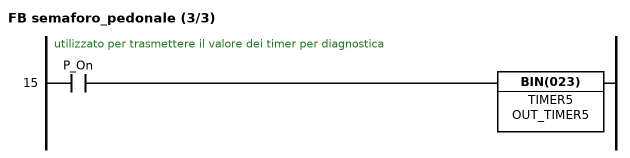
; [picture p24: FB semaforo_pedonale, rungs 15-15]
; rung 15: utilizzato per trasmettere il valore dei timer per diagnostica
LD P_On
BIN(023) TIMER5 OUT_TIMER5

## Function block stella_triangolo_MAT
VAR_INPUT
  start : BOOL;
  STOP : BOOL;
  ausiliario_K1 : BOOL;
  ausiliario_K2 : BOOL;
  ausiliario_K3 : BOOL;
  termica : BOOL;
  emergenza : BOOL;
END_VAR
VAR_OUTPUT
  linea : BOOL;
  stella : BOOL;
  triangolo : BOOL;
  lamp_blu : BOOL;
  lamp_verde1 : BOOL;
  lamp_verde2 : BOOL;
  lamp_gialla : BOOL;
  OUT_TIMER2 : WORD;
  OUT_TIMER1 : WORD;
END_VAR
VAR
  TIME : TIMER;
  err : BOOL;
END_VAR

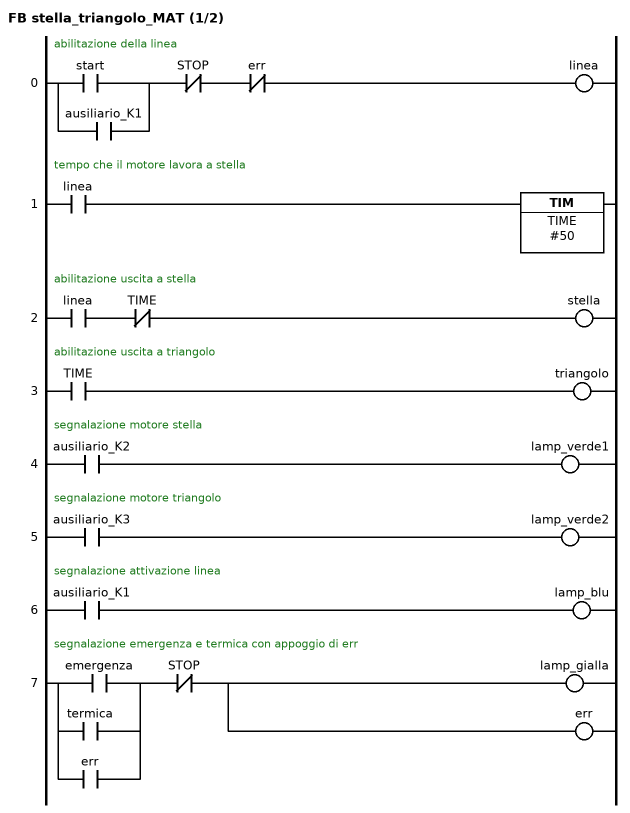
; rung 0: abilitazione della linea
LD start
OR ausiliario_K1
ANDNOT STOP
ANDNOT err
OUT linea
; rung 1: tempo che il motore lavora a stella
LD linea
TIM TIME #50
; rung 2: abilitazione uscita a stella
LD linea
ANDNOT TIME
OUT stella
; rung 3: abilitazione uscita a triangolo
LD TIME
OUT triangolo
; rung 4: segnalazione motore stella
LD ausiliario_K2
OUT lamp_verde1
; rung 5: segnalazione motore triangolo
LD ausiliario_K3
OUT lamp_verde2
; rung 6: segnalazione attivazione linea
LD ausiliario_K1
OUT lamp_blu
; rung 7: segnalazione emergenza e termica con appoggio di err
LD emergenza
OR termica
OR err
ANDNOT STOP
OUT lamp_gialla
OUT err

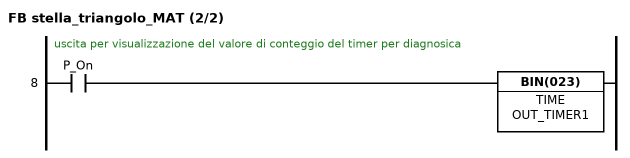
; rung 8: uscita per visualizzazione del valore di conteggio del timer per diagnosica
LD P_On
BIN(023) TIME OUT_TIMER1